// Mitsubishi GX Works2 project: com+   PLC: FX3U/FX3UC

// task Task_01 (event TRUE, interval 0, priority 31): POU_01

PROGRAM POU_01
MOV(MOV(MOV(MOV(M8411 ,H109F ,D8400),H11,D8401),K10,D8411),K80,D8411);

Y0:=NOT X1 AND (X0 OR (NOT X0 AND M0));

OUT_T( X2 OR (NOT X2 AND NOT X3 AND M1 ) ,TC0 , k30 );
OUT_T( X2 OR (NOT X2 AND NOT X3 AND M1 ) ,TC1 , k300 );
OUT_T( X3 OR (NOT X2 AND NOT X3 AND NOT  M1 ) ,TC2 , k30 );
OUT_T( X3 OR (NOT X2 AND NOT X3 AND NOT   M1 ) ,TC3 , k300 );
Y1:=NOT Y2 AND NOT X3  AND TS0   AND NOT  TS1;
Y2:=NOT Y1 AND NOT X2  AND TS2  AND NOT TS3 ;

Y3:=NOT X5 AND (X4 OR (NOT X4 AND M2));

OUT_T( X6 OR (NOT X6 AND NOT X7 AND M3 ) ,TC4 , k30 );
OUT_T( X6 OR (NOT X6 AND NOT X7 AND M3 ) ,TC5 , k300 );
OUT_T( X7 OR (NOT X6 AND NOT X7 AND NOT  M3 ) ,TC6 , k30 );
OUT_T( X7 OR (NOT X6 AND NOT X7 AND NOT   M3 ) ,TC7 , k300 );
Y4:=NOT Y5 AND NOT X7  AND TS4   AND NOT  TS5;
Y5:=NOT Y4 AND NOT X6  AND TS6  AND NOT TS7 ;

Y6:=NOT X11 AND (X10 OR (NOT X10 AND M4));

Y7:=NOT X13 AND (X12 OR (NOT X12 AND M5));

Y10:=NOT X15 AND (X14 OR (NOT X14 AND M6));

Y11:=NOT X17 AND (X16 OR (NOT X16 AND M7));

Y12:=NOT X21 AND (X20 OR (NOT X20 AND M8));

Y13:=NOT X23 AND (X22 OR (NOT X22 AND M9));

Y14:=NOT X25 AND (X24 OR (NOT X24 AND M10));

Y15:=NOT X27 AND (X26 OR (NOT X26 AND M11));

Y16:=NOT X31 AND (X30 OR (NOT X30 AND M12));

OUT_T( X32 OR (NOT X32 AND NOT X33 AND M13 ) ,TC8 , k30 );
OUT_T( X32 OR (NOT X32 AND NOT X33 AND M13 ) ,TC9 , k300 );
OUT_T( X33 OR (NOT X32 AND NOT X33 AND NOT  M13 ) ,TC10 , k30 );
OUT_T( X33 OR (NOT X32 AND NOT X33 AND NOT   M13 ) ,TC11 , k300 );
Y17:=NOT Y20 AND NOT X33  AND TS8   AND NOT  TS9;
Y20:=NOT Y17 AND NOT X32  AND TS10  AND NOT TS11 ;

OUT_T( X34 OR (NOT X34 AND NOT X35 AND M14 ) ,TC12 , k30 );
OUT_T( X34 OR (NOT X34 AND NOT X35 AND M14 ) ,TC13 , k300 );
OUT_T( X35 OR (NOT X34 AND NOT X35 AND NOT  M14 ) ,TC14 , k30 );
OUT_T( X35 OR (NOT X34 AND NOT X35 AND NOT   M14 ) ,TC15 , k300 );
Y21:=NOT Y22 AND NOT X35  AND TS12   AND NOT  TS13;
Y22:=NOT Y21 AND NOT X34  AND TS14  AND NOT TS15 ;

OUT_T( X36 OR (NOT X36 AND NOT X37 AND M15 ) ,TC16 , k30 );
OUT_T( X36 OR (NOT X36 AND NOT X37 AND M15 ) ,TC17 , k300 );
OUT_T( X37 OR (NOT X36 AND NOT X37 AND NOT  M15 ) ,TC18 , k30 );
OUT_T( X37 OR (NOT X36 AND NOT X37 AND NOT   M15 ) ,TC19 , k300 );
Y23:=NOT Y24 AND NOT X37  AND TS16   AND NOT  TS17;
Y24:=NOT Y23 AND NOT X36  AND TS18  AND NOT TS19 ;
END_PROGRAM
